// SIMATIC S7-200 project (STEP 7-Micro/WIN), CPU 226 CN REL 02.01

ORGANIZATION_BLOCK MAIN:OB1
TITLE=PROGRAM COMMENTS
BEGIN
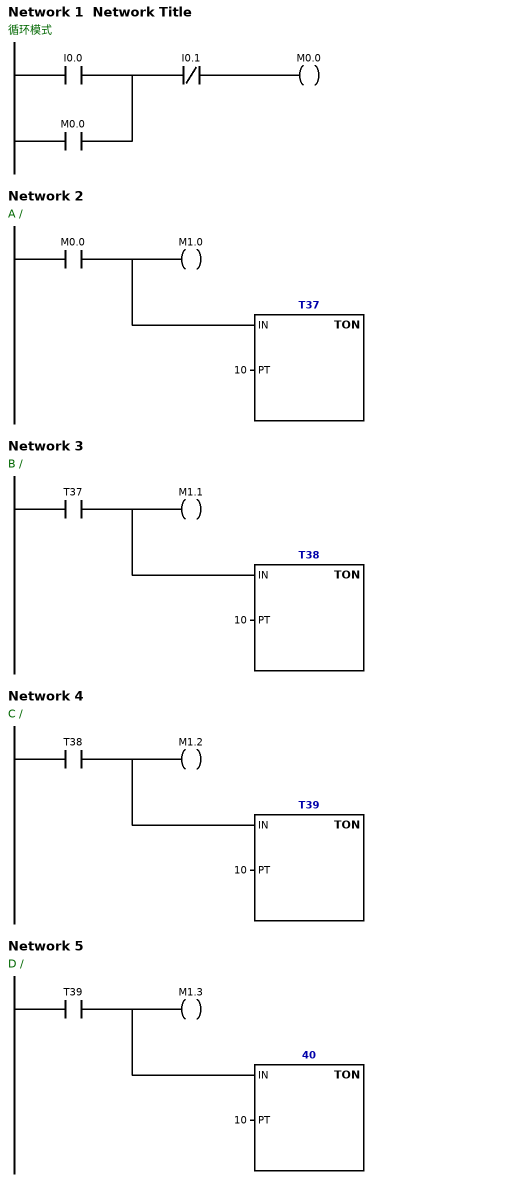
Network 1 // Network Title
// 循环模式
LD     I0.0
O      M0.0
AN     I0.1
=      M0.0
Network 2
// A
// 
LD     M0.0
=      M1.0
TON    T37, 10
Network 3
// B
// 
LD     T37
=      M1.1
TON    T38, 10
Network 4
// C
// 
LD     T38
=      M1.2
TON    T39, 10
Network 5
// D
// 
// (network saved uncompiled; LAD cells follow)
// row 0: c0 -| |- T39 v  c1 -( ) M1.3
// row 1: c0 ^  c1 --  c2 [TON 40 IN:=power@row1, PT:=10]
// row 2: c2 [box]
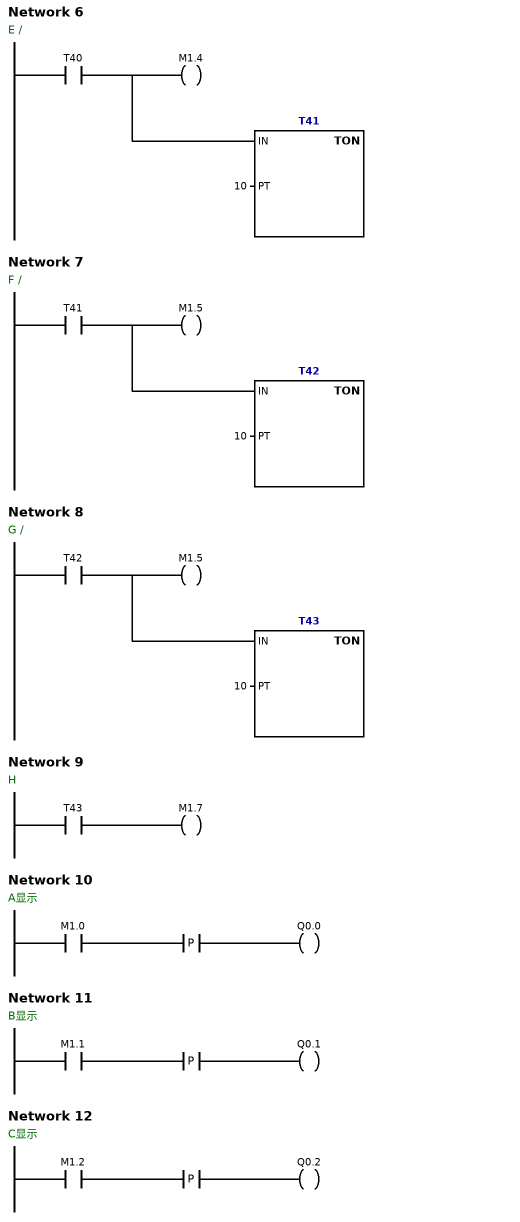
Network 6
// E
// 
LD     T40
=      M1.4
TON    T41, 10
Network 7
// F
// 
LD     T41
=      M1.5
TON    T42, 10
Network 8
// G
// 
LD     T42
=      M1.5
TON    T43, 10
Network 9
// H
LD     T43
=      M1.7
Network 10
// A显示
LD     M1.0
EU
=      Q0.0
Network 11
// B显示
LD     M1.1
EU
=      Q0.1
Network 12
// C显示
LD     M1.2
EU
=      Q0.2
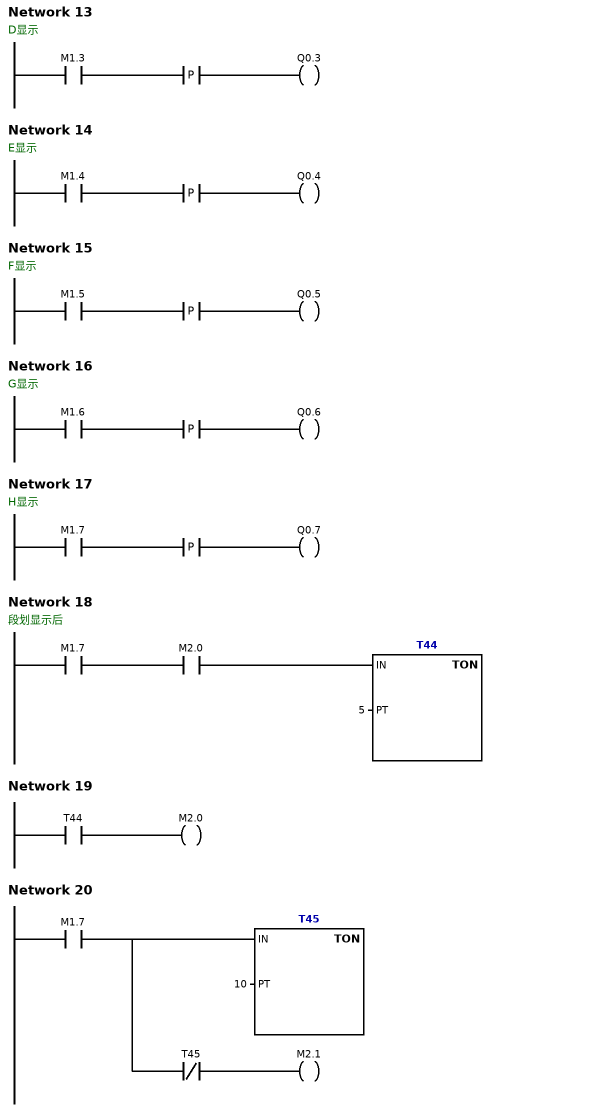
Network 13
// D显示
LD     M1.3
EU
=      Q0.3
Network 14
// E显示
LD     M1.4
EU
=      Q0.4
Network 15
// F显示
LD     M1.5
EU
=      Q0.5
Network 16
// G显示
LD     M1.6
EU
=      Q0.6
Network 17
// H显示
LD     M1.7
EU
=      Q0.7
Network 18
// 段划显示后
LD     M1.7
A      M2.0
TON    T44, 5
Network 19
LD     T44
=      M2.0
Network 20
LD     M1.7
TON    T45, 10
AN     T45
=      M2.1
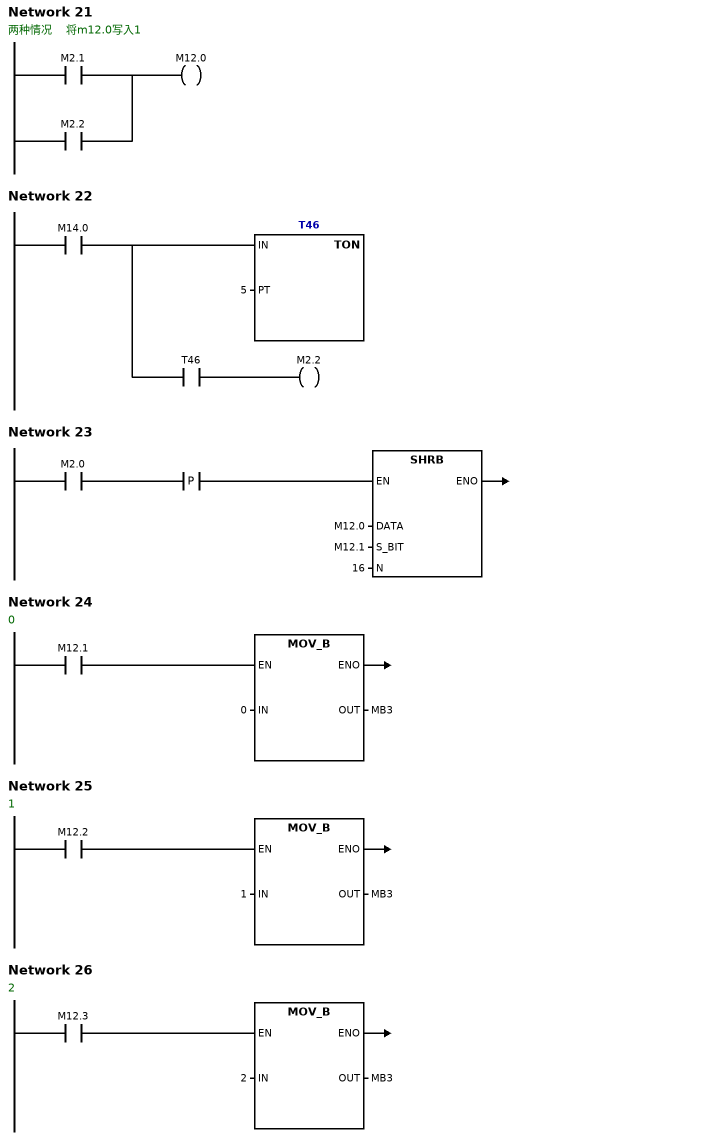
Network 21
// 两种情况    将m12.0写入1
LD     M2.1
O      M2.2
=      M12.0
Network 22
LD     M14.0
TON    T46, 5
A      T46
=      M2.2
Network 23
LD     M2.0
EU
SHRB   M12.0, M12.1, 16
Network 24
// 0
LD     M12.1
MOVB   0, MB3
Network 25
// 1
LD     M12.2
MOVB   1, MB3
Network 26
// 2
LD     M12.3
MOVB   2, MB3
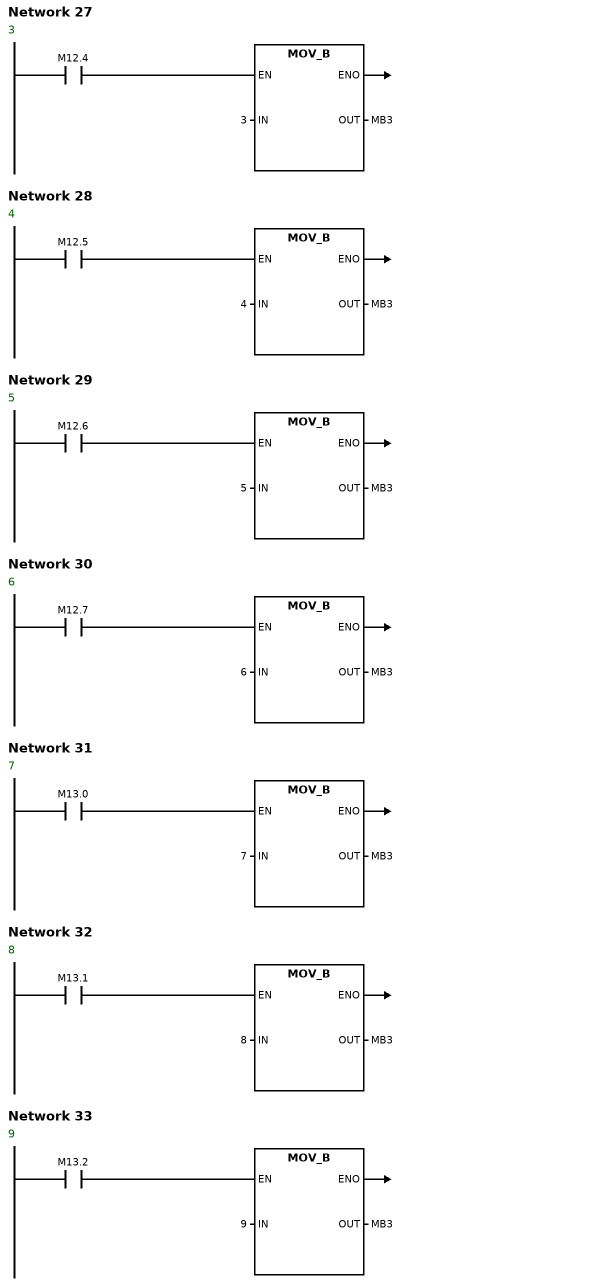
Network 27
// 3
LD     M12.4
MOVB   3, MB3
Network 28
// 4
LD     M12.5
MOVB   4, MB3
Network 29
// 5
LD     M12.6
MOVB   5, MB3
Network 30
// 6
LD     M12.7
MOVB   6, MB3
Network 31
// 7
LD     M13.0
MOVB   7, MB3
Network 32
// 8
LD     M13.1
MOVB   8, MB3
Network 33
// 9
LD     M13.2
MOVB   9, MB3
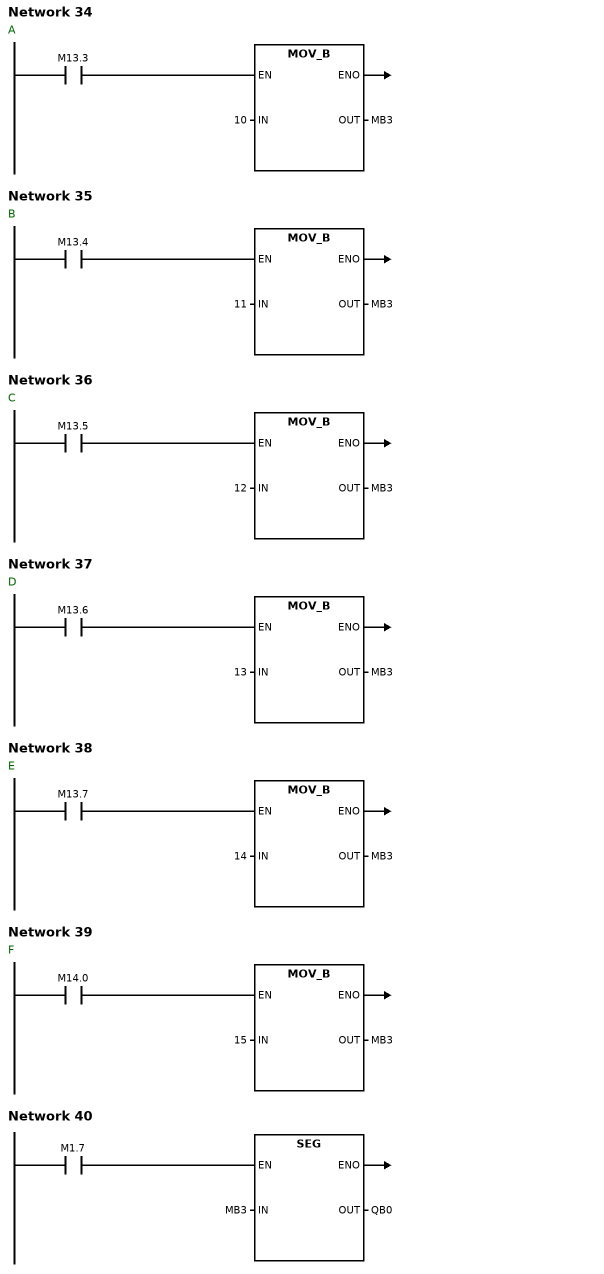
Network 34
// A
LD     M13.3
MOVB   10, MB3
Network 35
// B
LD     M13.4
MOVB   11, MB3
Network 36
// C
LD     M13.5
MOVB   12, MB3
Network 37
// D
LD     M13.6
MOVB   13, MB3
Network 38
// E
LD     M13.7
MOVB   14, MB3
Network 39
// F
LD     M14.0
MOVB   15, MB3
Network 40
LD     M1.7
SEG    MB3, QB0
END_ORGANIZATION_BLOCK
